PROGRAM MAIN
VAR
END_VAR

END_PROGRAM

(* stored: Version 1.1.0.1
   POU MAIN: Id {6318459e-7650-47dc-a61f-4823f2ea8bee} *)
